(* IEC 61131-3 sources: CodesysTest/alpha/export/FBs/Components/FunnelFB.pou/OpeningTime.prop, 1 file *)

(* ---- Set.pm.st ---- *)
(*#-#-#-#-#-#-#-#-#-#---Declaration---#-#-#-#-#-#-#-#-#-#-#-#-#*)

VAR
END_VAR
(*#-#-#-#-#-#-#-#-#-#---Implementation---#-#-#-#-#-#-#-#-#-#-#-#-#*)

openingTimer.PT := TO_TIME(OpeningTime * 1000);
